// TIA Portal V20 export
DATA_BLOCK "HMI_Interface_Parameter"   // DB262
// stored: Access Published, MemoryReserve 100
   VAR RETAIN
      ProcessUnitSelect : Int := 4;   // 1. Anode Reel Cut, 2. Cathode Reel Cut, 3. Stacking#1, 4.Stacking#2, 5. Inspection
   END_VAR
   VAR
      Recipe : "HMI_IF_Parameter_LIstRecipe_Interface";
      RecipeButton : "HMI_IF_Parameter_Save Button_UDT";
   END_VAR
   VAR RETAIN
      "Default Recipe" : "HMI_IF_Parameter_Recipe_Electrod_Interface";
      "Reelcut Recipe" { S7_SetPoint := 'True'} : "HMI_IF_Parameter_Recipe_Electrod_Reelcut_Interface";
      Parameter_Image : Array[0..17] of "HMI_IF_Parameter_Parameter_UDT";
      Parameter_Text : Array[0..154] of "HMI_IF_Parameter_Parameter_UDT";
      "Save Button" : "HMI_IF_Parameter_Save Button_UDT";
   END_VAR
   VAR
      "Save Button Old" { S7_SetPoint := 'True'} : "HMI_IF_Parameter_Save Button_UDT";
   END_VAR
   VAR RETAIN
      FATModeSelect : "LER_TypeFATMode_ModeSelect";
      FATModeInterface { S7_SetPoint := 'True'} : "LER_TypeFATModeInterface";
      VisionProgramNum : DWord;
   END_VAR
   VAR
      TempNull : Bool;
      TeachingPosIndex : SInt;
   END_VAR
   VAR RETAIN
      TeachingPosInterface : Array[0..48] of "LER_TypeTeachingPosInterface";
   END_VAR
   VAR
      PulseBit { ExternalAccessible := 'False'; ExternalVisible := 'False'; ExternalWritable := 'False'} : Array[0..99] of Bool;
   END_VAR
   VAR RETAIN
      Softcam : Array[0..48] of "LER_typeSoftCamRelation";
   END_VAR
   VAR
      SoftcamIndex : SInt;
   END_VAR
BEGIN
   // Parameter_Text[0] : CPM
   // Parameter_Text[2] : CellCount
   // Parameter_Text[6] : SleepModeActivationTime
   // Parameter_Text[7] : DeepSleepModeActivationTime
   // Parameter_Text[9] : Setpoint
   // Parameter_Text[10] : Kp
   // Parameter_Text[11] : Ki
   // Parameter_Text[13] : Pos1FinalRollerXFwdOutputCam
   // Parameter_Text[14] : Pos1FinalRollerXBwdOutputCam
   // Parameter_Text[15] : Pos1FinalRollerXStackTableDownOutputCam
   // Parameter_Text[16] : Pos1FinalRollerXStackAnodeVisionOutputCam
   // Parameter_Text[17] : Pos1FinalRollerXStackCathodeVisionOutputCam
   // Parameter_Text[18] : Pos1AnodePnPX1FwdOutputCam
   // Parameter_Text[19] : Pos1AnodePnPX1BwdOutputCam
   // Parameter_Text[20] : Pos1AnodePnPX1ReelCutDataDeleteOffOutputCam
   // Parameter_Text[21] : Pos1AnodePnPX2FwdOutputCam
   // Parameter_Text[22] : Pos1AnodePnPX2BwdOutputCam
   // Parameter_Text[23] : Pos1AnodePnPZ1Down1OutputCam
   // Parameter_Text[24] : Pos1AnodePnPZ1Up1OutputCam
   // Parameter_Text[25] : Pos1AnodePnPZ2Down1OutputCam
   // Parameter_Text[26] : Pos1AnodePnPZ2Up1OutputCam
   // Parameter_Text[27] : Pos1AnodePnPZ1Down2OutputCam
   // Parameter_Text[28] : Pos1AnodePnPZ1Up2OutputCam
   // Parameter_Text[29] : Pos1AnodePnPZ2Down2OutputCam
   // Parameter_Text[30] : Pos1AnodePnPZ2Up2OutputCam
   // Parameter_Text[31] : Pos1AnodePnPZ1SuctionOnOutputCam
   // Parameter_Text[32] : Pos1AnodePnPZ1SuctionOffOutputCam
   // Parameter_Text[33] : Pos1AnodePnPZ1ReelCutBlowOutputCam
   // Parameter_Text[34] : Pos1AnodePnPZ1ReelCutDataDeleteOnOutputCam
   // Parameter_Text[35] : Pos1AnodePnPZ1AlignVisionOutputCam
   // Parameter_Text[36] : Pos1AnodePnPZ2SuctionOnOutputCam
   // Parameter_Text[37] : Pos1AnodePnPZ2SuctionOffOutputCam
   // Parameter_Text[38] : Pos1AnodeAlignSuctionOnOutputCam
   // Parameter_Text[39] : Pos1AnodeAlignSuctionOffOutputCam
   // Parameter_Text[40] : Pos1CathodePnPX1FwdOutputCam
   // Parameter_Text[41] : Pos1CathodePnPX1BwdOutputCam
   // Parameter_Text[42] : Pos1CathodePnPX1ReelCutDataDeleteOffOutputCam
   // Parameter_Text[43] : Pos1CathodePnPX2FwdOutputCam
   // Parameter_Text[44] : Pos1CathodePnPX2BwdOutputCam
   // Parameter_Text[45] : Pos1CathodePnPZ1Down1OutputCam
   // Parameter_Text[46] : Pos1CathodePnPZ1Up1OutputCam
   // Parameter_Text[47] : Pos1CathodePnPZ2Down1OutputCam
   // Parameter_Text[48] : Pos1CathodePnPZ2Up1OutputCam
   // Parameter_Text[49] : Pos1CathodePnPZ1Down2OutputCam
   // Parameter_Text[50] : Pos1CathodePnPZ1Up2OutputCam
   // Parameter_Text[51] : Pos1CathodePnPZ2Down2OutputCam
   // Parameter_Text[52] : Pos1CathodePnPZ2Up2OutputCam
   // Parameter_Text[53] : Pos1CathodePnPZ1SuctionOnOutputCam
   // Parameter_Text[54] : Pos1CathodePnPZ1SuctionOffOutputCam
   // Parameter_Text[55] : Pos1CathodePnPZ1ReelCutBlowOutputCam
   // Parameter_Text[56] : Pos1CathodePnPZ1ReelCutDataDeleteOnOutputCam
   // Parameter_Text[57] : Pos1CathodePnPZ1AlignVisionOutputCam
   // Parameter_Text[58] : Pos1CathodePnPZ2SuctionOnOutputCam
   // Parameter_Text[59] : Pos1CathodePnPZ2SuctionOffOutputCam
   // Parameter_Text[60] : Pos1CathodeAlignSuctionOnOutputCam
   // Parameter_Text[61] : Pos1CathodeAlignSuctionOffOutputCam
   // Parameter_Text[62] : Pos2FinalRollerXFwdOutputCam
   // Parameter_Text[63] : Pos2FinalRollerXBwdOutputCam
   // Parameter_Text[64] : Pos2FinalRollerXStackTableDownOutputCam
   // Parameter_Text[65] : Pos2FinalRollerXStackAnodeVisionOutputCam
   // Parameter_Text[66] : Pos2FinalRollerXStackCathodeVisionOutputCam
   // Parameter_Text[67] : Pos2AnodePnPX1FwdOutputCam
   // Parameter_Text[68] : Pos2AnodePnPX1BwdOutputCam
   // Parameter_Text[69] : Pos2AnodePnPX1ReelCutDataDeleteOffOutputCam
   // Parameter_Text[70] : Pos2AnodePnPX2FwdOutputCam
   // Parameter_Text[71] : Pos2AnodePnPX2BwdOutputCam
   // Parameter_Text[72] : Pos2AnodePnPZ1Down1OutputCam
   // Parameter_Text[73] : Pos2AnodePnPZ1Up1OutputCam
   // Parameter_Text[74] : Pos2AnodePnPZ2Down1OutputCam
   // Parameter_Text[75] : Pos2AnodePnPZ2Up1OutputCam
   // Parameter_Text[76] : Pos2AnodePnPZ1Down2OutputCam
   // Parameter_Text[77] : Pos2AnodePnPZ1Up2OutputCam
   // Parameter_Text[78] : Pos2AnodePnPZ2Down2OutputCam
   // Parameter_Text[79] : Pos2AnodePnPZ2Up2OutputCam
   // Parameter_Text[80] : Pos2AnodePnPZ1SuctionOnOutputCam
   // Parameter_Text[81] : Pos2AnodePnPZ1SuctionOffOutputCam
   // Parameter_Text[82] : Pos2AnodePnPZ1ReelCutBlowOutputCam
   // Parameter_Text[83] : Pos2AnodePnPZ1ReelCutDataDeleteOnOutputCam
   // Parameter_Text[84] : Pos2AnodePnPZ1AlignVisionOutputCam
   // Parameter_Text[85] : Pos2AnodePnPZ2SuctionOnOutputCam
   // Parameter_Text[86] : Pos2AnodePnPZ2SuctionOffOutputCam
   // Parameter_Text[87] : Pos2AnodeAlignSuctionOnOutputCam
   // Parameter_Text[88] : Pos2AnodeAlignSuctionOffOutputCam
   // Parameter_Text[89] : Pos2CathodePnPX1FwdOutputCam
   // Parameter_Text[90] : Pos2CathodePnPX1BwdOutputCam
   // Parameter_Text[91] : Pos2CathodePnPX1ReelCutDataDeleteOffOutputCam
   // Parameter_Text[92] : Pos2CathodePnPX2FwdOutputCam
   // Parameter_Text[93] : Pos2CathodePnPX2BwdOutputCam
   // Parameter_Text[94] : Pos2CathodePnPZ1Down1OutputCam
   // Parameter_Text[95] : Pos2CathodePnPZ1Up1OutputCam
   // Parameter_Text[96] : Pos2CathodePnPZ2Down1OutputCam
   // Parameter_Text[97] : Pos2CathodePnPZ2Up1OutputCam
   // Parameter_Text[98] : Pos2CathodePnPZ1Down2OutputCam
   // Parameter_Text[99] : Pos2CathodePnPZ1Up2OutputCam
   // Parameter_Text[100] : Pos2CathodePnPZ2Down2OutputCam
   // Parameter_Text[101] : Pos2CathodePnPZ2Up2OutputCam
   // Parameter_Text[102] : Pos2CathodePnPZ1SuctionOnOutputCam
   // Parameter_Text[103] : Pos2CathodePnPZ1SuctionOffOutputCam
   // Parameter_Text[104] : Pos2CathodePnPZ1ReelCutBlowOutputCam
   // Parameter_Text[105] : Pos2CathodePnPZ1ReelCutDataDeleteOnOutputCam
   // Parameter_Text[106] : Pos2CathodePnPZ1AlignVisionOutputCam
   // Parameter_Text[107] : Pos2CathodePnPZ2SuctionOnOutputCam
   // Parameter_Text[108] : Pos2CathodePnPZ2SuctionOffOutputCam
   // Parameter_Text[109] : Pos2CathodeAlignSuctionOnOutputCam
   // Parameter_Text[110] : Pos2CathodeAlignSuctionOffOutputCam
   // Parameter_Text[111] : StageHeight
   // Parameter_Text[112] : StageGap
   // Parameter_Text[113] : FinalRollerStart
   // Parameter_Text[114] : FinalRollerEnd
   // Parameter_Text[115] : PnPXStart
   // Parameter_Text[116] : PnPXEnd
   // Parameter_Text[117] : PnPZDownStart
   // Parameter_Text[118] : PnPZDownEnd
   // Parameter_Text[119] : PnPZUpStart
   // Parameter_Text[120] : PnPZUpEnd
   // Parameter_Text[121] : MandrelBwdStart
   // Parameter_Text[122] : MandrelBwdEnd
   // Parameter_Text[123] : MandrelFwdStart
   // Parameter_Text[124] : MandrelFwdEnd
   // Parameter_Text[125] : MandrelUpStart1
   // Parameter_Text[126] : MandrelUpEnd1
   // Parameter_Text[127] : MandrelUpStart2
   // Parameter_Text[128] : MandrelUpEnd2
   // Parameter_Text[129] : MandrelDownStart
   // Parameter_Text[130] : MandrelDownEnd
   // Parameter_Text[131] : MandrelYTerm
   // Parameter_Text[132] : MandrelZTerm
   // Parameter_Text[133] : MandrelBwdOffset
   // Parameter_Text[134] : MandrelFwdOffset
   // Parameter_Text[135] : FinalRollerStart
   // Parameter_Text[136] : FinalRollerEnd
   // Parameter_Text[137] : PnPXStart
   // Parameter_Text[138] : PnPXEnd
   // Parameter_Text[139] : PnPZDownStart
   // Parameter_Text[140] : PnPZDownEnd
   // Parameter_Text[141] : PnPZUpStart
   // Parameter_Text[142] : PnPZUpEnd
   // Parameter_Text[143] : MandrelBwdStart
   // Parameter_Text[144] : MandrelBwdEnd
   // Parameter_Text[145] : MandrelFwdStart
   // Parameter_Text[146] : MandrelFwdEnd
   // Parameter_Text[147] : MandrelUpStart1
   // Parameter_Text[148] : MandrelUpEnd1
   // Parameter_Text[149] : MandrelUpStart2
   // Parameter_Text[150] : MandrelUpEnd2
   // Parameter_Text[151] : MandrelDownStart
   // Parameter_Text[152] : MandrelDownEnd
   // Parameter_Text[153] : FinalRollerBwdPos
   // Parameter_Text[154] : FinalRollerFwdPos
END_DATA_BLOCK
